ADAPTER IDischargeStatus (* Adapter Interface *)
  (* Standard: 61499-1 *)
  (* Version 0.0, 6/8/2026, Schneider Electric *)
  PACKAGE SE.Nereda;
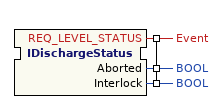
  EVENT_OUTPUT
    REQ_LEVEL_STATUS WITH Aborted, Interlock;
  END_EVENT
  VAR_OUTPUT
    Aborted : BOOL;
    Interlock : BOOL;
  END_VAR
  SERVICE SOCKET/PLUG
    SEQUENCE request_confirm
      SOCKET.REQ(REQD) -> PLUG.REQ(REQD);
      PLUG.CNF(CNFD) -> SOCKET.CNF(CNFD);
    END_SEQUENCE
    SEQUENCE indication_response
      PLUG.IND(INDD) -> SOCKET.IND(INDD);
      SOCKET.RSP(RSPD) -> PLUG.RSP(RSPD);
    END_SEQUENCE
  END_SERVICE
END_ADAPTER
